// TwinCAT 3 PLC project test
// libraries:
//   Tc2_Standard, * (Beckhoff Automation GmbH)
//   Tc2_System, * (Beckhoff Automation GmbH)
//   Tc3_Interfaces, * (Beckhoff Automation GmbH)
//   Tc3_Module, * (Beckhoff Automation GmbH)
// project tree:
//   Data types/ MyStruct.TcDUT
//   Global Variables/ Global_Variables.TcGVL, Variable_Configuration.TcGVL
//   POUs/ MAIN.TcPOU
//   / Standard.TcTTO
// real-time tasks:
//   TASK PlcTask: cycle T#10ms, priority 20, ADS port 350
//   TASK fast: cycle T#1ms, priority 21, ADS port 351
//   TASK medium: cycle T#1ms, priority 22, ADS port 352
//   TASK slow: cycle T#100000us, priority 23, ADS port 353

CONFIGURATION test
    RESOURCE PLC ON TwinCAT3
        TASK Standard(INTERVAL := T#10ms, PRIORITY := 20);
        PROGRAM MAIN WITH Standard : MAIN;
    END_RESOURCE
END_CONFIGURATION

// ---- Data types/MyStruct.TcDUT
TYPE MyStruct :
STRUCT
	myInt: INT := 1;
	myBool: BOOL := FALSE;	
END_STRUCT
END_TYPE

// ---- Global Variables/Global_Variables.TcGVL
{attribute 'Tc2GvlVarNames'}
VAR_GLOBAL
END_VAR

// ---- Global Variables/Variable_Configuration.TcGVL
{attribute 'Tc2GvlVarNames'}
VAR_CONFIG
END_VAR

// ---- POUs/MAIN.TcPOU
PROGRAM MAIN
VAR
	var1: INT;
	var2: STRING(80) := 'This is a default value';
	var3: INT := 0;
	var4: INT := 0;
	var5: MyStruct;
	var6: MyStruct;

	counter: INT := 0;
END_VAR

var1 := var1 + 3;

counter := counter + 1;

IF counter = 100 THEN
	counter := 0;
	var4 := var4 + 1;
	var5.myBool := NOT var5.myBool;
	var5.myInt := var5.myInt + 1;
END_IF

END_PROGRAM
